// TIA Portal V20 export
TYPE "LConSMC_typeKpAdaptionOutput"
// stored: Access Published
   STRUCT
      busy : Bool;   // TRUE: Funktionsblock ist aktiv / TRUE: Function block is in operation
      kpAdaptionValue : Real;   // [0-100%] Adaptionswert Dieser Wert wird mit dem Kp des Drehzahlreglers multipliziert / [0-100%] Adaption value This value will be multiplied with the speed controler Kp value
      error : Bool;   // TRUE: Ein Fehler ist aufgetreten / TRUE: Error has occured
      errorID : DWord;   // Detaillierte Fehlerbeschreibung / Detailed error description
   END_STRUCT;
END_TYPE
